KUKA KRL program: wkz2_ab.src, wkz2_ab.dat

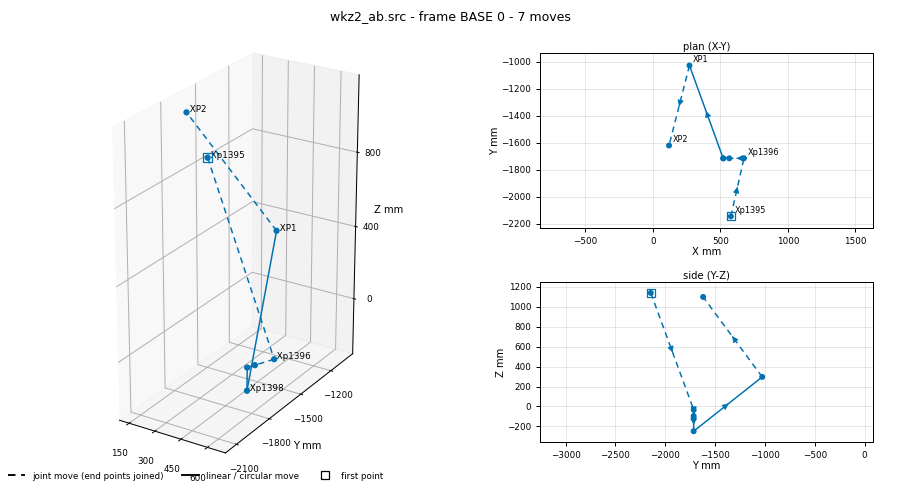
[picture p0: tool path of wkz2_ab.src in frame BASE 0, 7 of 7 moves have a stored position in this frame; points joined in program order, loops and branches not executed]
--- wkz2_ab.src ---
&ACCESS RVO2
&REL 152
&COMMENT Entrega X1
DEF WKZ2_AB ( )
  ;FOLD INI;%{PE}%V2.2.2,%MKUKATPBASIS,%CINIT,%VCOMMON,%P
  ;FOLD BAS INI;%{PE}%V2.2.2,%MKUKATPBASIS,%CINIT,%VINIT,%P
  INTERRUPT DECL 3 WHEN $STOPMESS==TRUE DO IR_STOPM ( )
  INTERRUPT ON 3
  BAS (#INITMOV,0 )
  ;ENDFOLD
  ;FOLD A20 INI;%{E}%V2.2.2,%MKUKATPA20,%CINIT,%VINIT,%P
  IF ARC20==TRUE THEN
    A20 (ARC_INI)
    INTERRUPT DECL 6 WHEN $CYCFLAG[3]==FALSE DO A20(TECH_STOP2)
  ENDIF
  ;ENDFOLD
  ;FOLD A10 INI;%{E}%V2.2.2,%MKUKATPARC,%CINIT,%VINIT,%P
  IF A10_OPTION==#ACTIVE THEN
    INTERRUPT DECL 4 WHEN $CYCFLAG[2]==FALSE DO A10 (#APPL_ERROR)
    INTERRUPT DECL 7 WHEN A_ARC_SWI==#ACTIVE DO A10 (#ARC_SEAM)
    INTERRUPT DECL 5 WHEN A_FLY_ARC==TRUE DO A10 (#HPU_ARC)
    INTERRUPT  ON 5
    A10_INI ( )
  ENDIF
  ;ENDFOLD
  ;FOLD GRIPPER INI;%{E}%V2.2.2,%MKUKATPGRIPPER,%CINIT,%VINIT,%P
  USER_GRP(0,DUMMY,DUMMY,GDEFAULT)
  ;ENDFOLD
  ;FOLD SPOT INI;%{E}%V.2.2,%MKUKATPSPOT,%CINIT,%VINIT,%P

  ;ENDFOLD
  ;FOLD TOUCHSENSE INI;%{E}%V2.2.2,%MKUKATPTS,%CINIT,%VINIT,%P
  IF H70_OPTION THEN
    INTERRUPT DECL 15 WHEN $MEAS_PULSE[TOUCH_I[TOUCH_ACTIVE].IN_NR] DO H70 (6,CD0 )
    INTERRUPT DECL 16 WHEN $ZERO_MOVE DO H70 (7,CD0 )
    INTERRUPT DECL 17 WHEN $TECHPAR_C[FG_TOUCH,8]>0.5 DO H70 (8,CD0)
    H70 (1,CD0 )
  ENDIF
  ;ENDFOLD
  ;FOLD USER INI;%{P}%V2.2.2,%MKUKATPUSER,%CINIT,%VINIT,%P
  ;Make your modifications here
  ;ENDFOLD
  ;ENDFOLD

; Caracterização dos meios de produção: P13.060-R4
; Versão atual: 20/07/2013 12:00  Nome: Deposita pinça X1
; Magazine

chk_w2_wechs_ok ( )     ; VERIFICAÇÃO DE FERRAMENTA: X1

;FOLD PULSE 167 'protecao da pinca abrir'  State= TRUE CONT  Time= 1 sec;%{PE}%R 4.1.16,%MKUKATPBASIS,%COUT,%VPULSE,%P 2:167, 3:'protecao da pinca abrir', 5:TRUE, 6:CONTINUE, 8:1
CONTINUE
PULSE($OUT[167], TRUE,1)
;ENDFOLD
;FOLD WAIT FOR IN 219 'placas de suporte fundidas'  State= TRUE ;%{PE}%R 4.1.16,%MKUKATPBASIS,%CWAIT_FOR,%VWAIT_FOR,%P 1:0, 2:219, 3:'placas de suporte fundidas', 5:TRUE, 6:
WAIT FOR $IN[219]==TRUE
;ENDFOLD
;FOLD WAIT FOR IN 161 'deposito ocupado'  State= FALSE ;%{PE}%R 4.1.16,%MKUKATPBASIS,%CWAIT_FOR,%VWAIT_FOR,%P 1:0, 2:161, 3:'deposito ocupado', 5:FALSE, 6:
WAIT FOR $IN[161]==FALSE
;ENDFOLD
;FOLD WAIT FOR IN 165 'protecao de pinca aberto'  State= TRUE ;%{PE}%R 4.1.16,%MKUKATPBASIS,%CWAIT_FOR,%VWAIT_FOR,%P 1:0, 2:165, 3:'protecao de pinca aberto', 5:TRUE, 6:
WAIT FOR $IN[165]==TRUE
;ENDFOLD
;FOLD WAIT FOR IN 166 'protecao de pinca fechado'  State= FALSE ;%{PE}%R 4.1.16,%MKUKATPBASIS,%CWAIT_FOR,%VWAIT_FOR,%P 1:0, 2:166, 3:'protecao de pinca fechado', 5:FALSE, 6:
WAIT FOR $IN[166]==FALSE
;ENDFOLD

;FOLD PTP p1395 CONT Vel= 80 % P_OLP3 Tool[2]:GUN X1 Base[0];%{PE}%R 4.1.16,%MKUKATPBASIS,%CMOVE,%VPTP,%P 1:PTP, 2:p1395, 3:C_PTP, 5:80, 7:P_OLP3
$BWDSTART = FALSE
PDAT_ACT=PP_OLP3
BAS(#PTP_DAT)
FDAT_ACT=Fp1395
BAS(#FRAMES)
BAS(#VEL_PTP,80)
PTP Xp1395 C_PTP
;ENDFOLD

;FOLD PTP p1396 CONT Vel= 100 % PDAT3 Tool[2]:GUN X1 Base[0];%{PE}%R 4.1.16,%MKUKATPBASIS,%CMOVE,%VPTP,%P 1:PTP, 2:p1396, 3:C_PTP, 5:100, 7:PDAT3
$BWDSTART = FALSE
PDAT_ACT=PPDAT3
BAS(#PTP_DAT)
FDAT_ACT=Fp1396
BAS(#FRAMES)
BAS(#VEL_PTP,100)
PTP Xp1396 C_PTP
;ENDFOLD
;FOLD PTP P3 CONT Vel= 100 % PDAT4 Tool[2]:GUN X1 Base[0];%{PE}%R 4.1.16,%MKUKATPBASIS,%CMOVE,%VPTP,%P 1:PTP, 2:P3, 3:C_PTP, 5:100, 7:PDAT4
$BWDSTART = FALSE
PDAT_ACT=PPDAT4
BAS(#PTP_DAT)
FDAT_ACT=FP3
BAS(#FRAMES)
BAS(#VEL_PTP,100)
PTP XP3 C_PTP
;ENDFOLD
;FOLD LIN p1397  Vel= 0.4 m/s L_OLP2 Tool[2]:GUN X1 Base[0];%{PE}%R 4.1.16,%MKUKATPBASIS,%CMOVE,%VLIN,%P 1:LIN, 2:p1397, 3:, 5:0.4, 7:L_OLP2
$BWDSTART = FALSE
LDAT_ACT=LL_OLP2
BAS(#CP_DAT)
FDAT_ACT=Fp1397
BAS(#FRAMES)
BAS(#VEL_CP,0.4)
LIN Xp1397
;ENDFOLD

$advance=0

;FOLD ; posicao de deposito;%{PE}%R 4.1.16,%MKUKATPBASIS,%CCOMMENT,%VNORMAL,%P 2:posicao de deposito
;ENDFOLD
;FOLD LIN p1398  Vel= 0.25 m/s CPDAT2 Tool[2]:GUN X1 Base[0];%{PE}%R 4.1.16,%MKUKATPBASIS,%CMOVE,%VLIN,%P 1:LIN, 2:p1398, 3:, 5:0.25, 7:CPDAT2
$BWDSTART = FALSE
LDAT_ACT=LCPDAT2
BAS(#CP_DAT)
FDAT_ACT=Fp1398
BAS(#FRAMES)
BAS(#VEL_CP,0.25)
LIN Xp1398
;ENDFOLD

;FOLD IBUS  OFF;%{PE}%R 4.1.16,%MKUKATPBASIS,%CIBUS,%VMAP,%P 2:#OFF, 3:1
$IBUS_OFF=$IBUS_ON
$IBUS_ON=0
;ENDFOLD
;FOLD WAIT FOR IN 161 'deposito ocupado'  State= TRUE ;%{PE}%R 4.1.16,%MKUKATPBASIS,%CWAIT_FOR,%VWAIT_FOR,%P 1:0, 2:161, 3:'deposito ocupado', 5:TRUE, 6:
WAIT FOR $IN[161]==TRUE
;ENDFOLD
;FOLD OUT 224 'Bloqueio MPS'  State= FALSE ;%{PE}%R 4.1.16,%MKUKATPBASIS,%COUT,%VOUTX,%P 2:224, 3:'Bloqueio MPS', 5:FALSE, 6:
$OUT[224]=FALSE
;ENDFOLD
;FOLD OUT 223 'Desbloqueio MPS'  State= TRUE ;%{PE}%R 4.1.16,%MKUKATPBASIS,%COUT,%VOUTX,%P 2:223, 3:'Desbloqueio MPS', 5:TRUE, 6:
$OUT[223]=TRUE
;ENDFOLD
;FOLD WAIT FOR IN 217 'MPS destravado'  State= TRUE ;%{PE}%R 4.1.16,%MKUKATPBASIS,%CWAIT_FOR,%VWAIT_FOR,%P 1:0, 2:217, 3:'MPS destravado', 5:TRUE, 6:
WAIT FOR $IN[217]==TRUE
;ENDFOLD
;FOLD WAIT FOR IN 221 'MPS travado'  State= FALSE ;%{PE}%R 4.1.16,%MKUKATPBASIS,%CWAIT_FOR,%VWAIT_FOR,%P 1:0, 2:221, 3:'MPS travado', 5:FALSE, 6:
WAIT FOR $IN[221]==FALSE
;ENDFOLD
;FOLD WAIT Time= 1 sec;%{PE}%R 4.1.16,%MKUKATPBASIS,%CWAIT,%VWAIT,%P 2:1
WAIT SEC 1
;ENDFOLD
;FOLD WAIT FOR IN 217 'MPS Destravado'  State= TRUE ;%{PE}%R 4.1.16,%MKUKATPBASIS,%CWAIT_FOR,%VWAIT_FOR,%P 1:0, 2:217, 3:'MPS Destravado', 5:TRUE, 6:
WAIT FOR $IN[217]==TRUE
;ENDFOLD

;FOLD LIN P1  Vel= 0.3 m/s CPDAT1 Tool[8]:Tool changer Base[0];%{PE}%R 4.1.16,%MKUKATPBASIS,%CMOVE,%VLIN,%P 1:LIN, 2:P1, 3:, 5:0.3, 7:CPDAT1
$BWDSTART = FALSE
LDAT_ACT=LCPDAT1
BAS(#CP_DAT)
FDAT_ACT=FP1
BAS(#FRAMES)
BAS(#VEL_CP,0.3)
LIN XP1
;ENDFOLD

;FOLD WAIT FOR IN 219 'placas de suporte fundidas'  State= FALSE ;%{PE}%R 4.1.16,%MKUKATPBASIS,%CWAIT_FOR,%VWAIT_FOR,%P 1:0, 2:219, 3:'placas de suporte fundidas', 5:FALSE, 6:
WAIT FOR $IN[219]==FALSE
;ENDFOLD
;FOLD WAIT FOR IN 161 'deposito ocupado'  State= TRUE ;%{PE}%R 4.1.16,%MKUKATPBASIS,%CWAIT_FOR,%VWAIT_FOR,%P 1:0, 2:161, 3:'deposito ocupado', 5:TRUE, 6:
WAIT FOR $IN[161]==TRUE
;ENDFOLD
;FOLD OUT 223 'Desbloqueio MPS'  State= FALSE ;%{PE}%R 4.1.16,%MKUKATPBASIS,%COUT,%VOUTX,%P 2:223, 3:'Desbloqueio MPS', 5:FALSE, 6:
$OUT[223]=FALSE
;ENDFOLD

;FOLD PTP P2  Vel= 100 % PDAT2 Tool[8]:Tool changer Base[0];%{PE}%R 4.1.16,%MKUKATPBASIS,%CMOVE,%VPTP,%P 1:PTP, 2:P2, 3:, 5:100, 7:PDAT2
$BWDSTART = FALSE
PDAT_ACT=PPDAT2
BAS(#PTP_DAT)
FDAT_ACT=FP2
BAS(#FRAMES)
BAS(#VEL_PTP,100)
PTP XP2
;ENDFOLD

;FOLD OUT 840 'R4 solda geometri concluida'  State= FALSE ;%{PE}%R 4.1.16,%MKUKATPBASIS,%COUT,%VOUTX,%P 2:840, 3:'R4 solda geometri concluida', 5:FALSE, 6:
$OUT[840]=FALSE
;ENDFOLD
;FOLD PULSE 168 'protecao da pinca fechar'  State= TRUE   Time= 1 sec;%{PE}%R 4.1.16,%MKUKATPBASIS,%COUT,%VPULSE,%P 2:168, 3:'protecao da pinca fechar', 5:TRUE, 6:, 8:1
PULSE($OUT[168], TRUE,1)
;ENDFOLD

END

--- wkz2_ab.dat ---
&ACCESS RVO2
&REL 152
&COMMENT Entrega X1
DEFDAT  WKZ2_AB
;FOLD EXTERNAL DECLARATIONS;%{PE}%V2.2.2,%MKUKATPBASIS,%CEXT,%VCOMMON,%P
;FOLD BAS EXT;%{PE}%V2.2.2,%MKUKATPBASIS,%CEXT,%VEXT,%P
EXT  BAS (BAS_COMMAND  :IN,REAL  :IN )
DECL INT SUCCESS
;ENDFOLD
;FOLD A10 EXT;%{E}%V2.2.2,%MKUKATPARC,%CEXT,%VEXT,%P
EXT  A10 (A_CMD_T  :IN,A_STRT_T  :IN,A_WELD_T  :IN,A_END_T  :IN,INT  :IN )
;ENDFOLD
;FOLD A20 EXT;%{E}%V2.2.2,%MKUKATPA20,%CEXT,%VEXT,%P
EXT  A20 (INT  :IN,WELD_ST  :IN,WELD_FI  :IN,INT  :IN )
;ENDFOLD
;FOLD GRIPPER EXT;%{E}%V2.2.2,%MKUKATPGRIPPER,%CEXT,%VEXT,%P
EXT  H50 (INT  :IN,INT  :IN,INT  :IN,GRP_TYP  :IN )
;ENDFOLD
;FOLD SPOT EXT;%{E}%V2.2.2,%MKUKATPSPOT,%CEXT,%VEXT,%P
EXT  USERSPOT (S_COMMAND  :IN,SPOT_TYPE  :IN )
;ENDFOLD
;FOLD TOUCHSENSE EXT;%{E}%V2.2.2,%MKUKATPTS,%CEXT,%VEXT,%P
EXT  H70 (INT  :IN,SRCH_TYP_2  :OUT,E6POS  :IN,SRCH_TYP_3  :IN,SRCH_TYP_2  :IN,SRCH_TYP_2  :IN,SRCH_TYP_2  :IN,SRCH_TYP_2  :IN,SRCH_TYP_2  :IN,INT  :IN )
;ENDFOLD
;FOLD USER EXT;%{}%V2.2.2,%MKUKATPUSER,%CEXT,%VEXT,%P
;Make here your modifications
;ENDFOLD
;ENDFOLD

;# ============ START PATH : za_p13060r4_x1 =============
DECL FDAT Fp1395={TOOL_NO 2,BASE_NO 0,IPO_FRAME #BASE}
DECL PDAT PP_OLP3={VEL 100.0,ACC 100.0,APO_DIST 100.0}
DECL E6POS Xp1395={x 577.786194,y -2145.35303,z 1139.39697,a -103.128304,b -38.1844902,c -131.547501,s 2,t 34,e1 0.0,e2 0.0,e3 0.0,e4 0.0,e5 0.0,e6 0.0}
DECL FDAT Fp1396={TOOL_NO 2,BASE_NO 0,IPO_FRAME #BASE}
DECL E6POS Xp1396={x 674.980286,y -1714.73901,z -33.193409,a -89.925621,b -0.0332944803,c -150.488693,s 2,t 34,e1 0.0,e2 0.0,e3 0.0,e4 0.0,e5 0.0,e6 0.0}
DECL LDAT LL_OLP1={VEL 0.25,ACC 100.0,APO_DIST 0.0,APO_FAC 0.0}
DECL FDAT Fp1397={TOOL_NO 2,BASE_NO 0,IPO_FRAME #BASE}
DECL E6POS Xp1397={x 522.117798,y -1715.25903,z -119.689102,a -89.9201965,b -0.0407406501,c -150.485199,s 2,t 34,e1 0.0,e2 0.0,e3 0.0,e4 0.0,e5 0.0,e6 0.0}
DECL LDAT LL_OLP2={VEL 0.25,ACC 100.0,APO_DIST 0.0,APO_FAC 0.0}
DECL FDAT Fp1398={TOOL_NO 2,BASE_NO 0,IPO_FRAME #BASE}
DECL E6POS Xp1398={x 521.015686,y -1715.33997,z -247.871796,a -89.9215622,b -0.0402558111,c -150.485199,s 2,t 34,e1 0.0,e2 0.0,e3 0.0,e4 0.0,e5 0.0,e6 0.0}
DECL BASIS_SUGG_T LAST_BASIS={POINT1[] "P3                      ",POINT2[] "P3                      ",CP_PARAMS[] "CPDAT1                  ",PTP_PARAMS[] "PDAT4                   ",CONT[] "C_PTP                   ",CP_VEL[] "2                       ",PTP_VEL[] "100                     "}
DECL E6POS XP1={x 270.879211,y -1027.302,z 296.65271,a 0.0800363123,b 0.485235304,c 179.9599,s 2,t 34,e1 0.0,e2 0.0,e3 0.0,e4 0.0,e5 0.0,e6 0.0}
DECL FDAT FP1={TOOL_NO 8,BASE_NO 0,IPO_FRAME #BASE}
DECL LDAT LCPDAT1={VEL 2.0,ACC 100.0,APO_DIST 100.0,APO_FAC 50.0}
DECL LDAT LCPDAT2={VEL 2.0,ACC 100.0,APO_DIST 100.0,APO_FAC 50.0}
DECL E6POS XP2={x 119.392197,y -1620.22205,z 1099.026,a -26.99893,b -12.1279402,c 123.912697,s 2,t 34,e1 0.0,e2 0.0,e3 0.0,e4 0.0,e5 0.0,e6 0.0}
DECL FDAT FP2={TOOL_NO 8,BASE_NO 0,IPO_FRAME #BASE}
DECL PDAT PPDAT2={VEL 100.0,ACC 100.0,APO_DIST 100.0}
DECL PDAT PPDAT3={VEL 100.0,ACC 100.0,APO_DIST 30.0}
DECL E6POS XP3={x 565.923218,y -1715.12805,z -94.888443,a -89.9212418,b -0.0401239395,c -150.485794,s 2,t 34,e1 0.0,e2 0.0,e3 0.0,e4 0.0,e5 0.0,e6 0.0}
DECL FDAT FP3={TOOL_NO 2,BASE_NO 0,IPO_FRAME #BASE}
DECL PDAT PPDAT4={VEL 100.0,ACC 100.0,APO_DIST 10.0}
ENDDAT
